FUNCTION_BLOCK FB_RetrocederPlato_SFC
VAR_IN_OUT
	   TpoEmpujadorAvanza: TIME;
END_VAR

VAR_INPUT
    // SFC-Flags
    SFCPause: BOOL;
    SFCReset: BOOL;
    
    // Indicadores de sincronizacion
    Ack: BOOL := TRUE;
    Execute: BOOL;
    
    // Entradas
   PlatoEmpujadorDetras : BOOL;
END_VAR
VAR_OUTPUT
    // Indicadores de sincronizacion
    Done: BOOL;
    Ready: BOOL;
    
    // Salidas
    PlatoEmpujadorAvanza : BOOL;
	PlatoRetenedorAtras : BOOL;
END_VAR
VAR
	S3: INT;
END_VAR

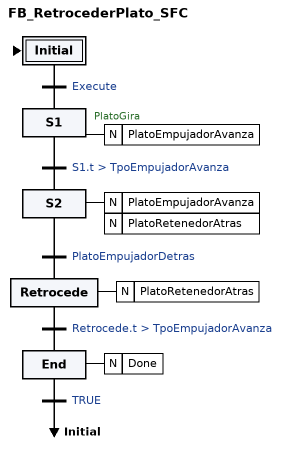
INITIAL_STEP Initial:
END_STEP
TRANSITION FROM Initial TO S1
    := Execute;
END_TRANSITION
// PlatoGira
STEP S1:
    PlatoEmpujadorAvanza(N);
END_STEP
TRANSITION FROM S1 TO S2
    := S1.t > TpoEmpujadorAvanza;
END_TRANSITION
STEP S2:
    PlatoEmpujadorAvanza(N);
    PlatoRetenedorAtras(N);
END_STEP
TRANSITION FROM S2 TO Retrocede
    := PlatoEmpujadorDetras;
END_TRANSITION
STEP Retrocede:
    PlatoRetenedorAtras(N);
END_STEP
TRANSITION FROM Retrocede TO End
    := Retrocede.t > TpoEmpujadorAvanza;
END_TRANSITION
STEP End:
    Done(N);
END_STEP
TRANSITION FROM End TO Initial
    := TRUE;
END_TRANSITION

END_FUNCTION_BLOCK

(* stored: Version 1.1.0.1, ProductVersion 3.1.4024.9
   POU FB_RetrocederPlato_SFC: Id {6a40a4e0-f3e4-494f-8d61-61468e6e5e1d}, SpecialFunc None *)
